// TIA Portal V20 export
FUNCTION "Scaling_pls_angle" : Void   // FC12, LAD
// stored: Namespace Global, SetENOAutomatically false
   VAR_INPUT
      "I_angle target" : Int;
      "I_angle min" : Int;
      "I_angle max" : Int;
      "I_pulse min" : Int;
      "I_pulse max" : Int;
   END_VAR
   VAR_OUTPUT
      "pulse target low" : Byte;
      "pulse target high" : Byte;
   END_VAR
   VAR_TEMP
      R_pulse_calcul : Real;
      R_angle_calcul : Real;
      pulse_target_int : Int;
      Int4 : Int;
      Int5 : Int;
      Real1 : Real;
      Real2 : Real;
      Real3 : Real;
      Real4 : Real;
   END_VAR
BEGIN

REGION Network 1: Convert diff in real
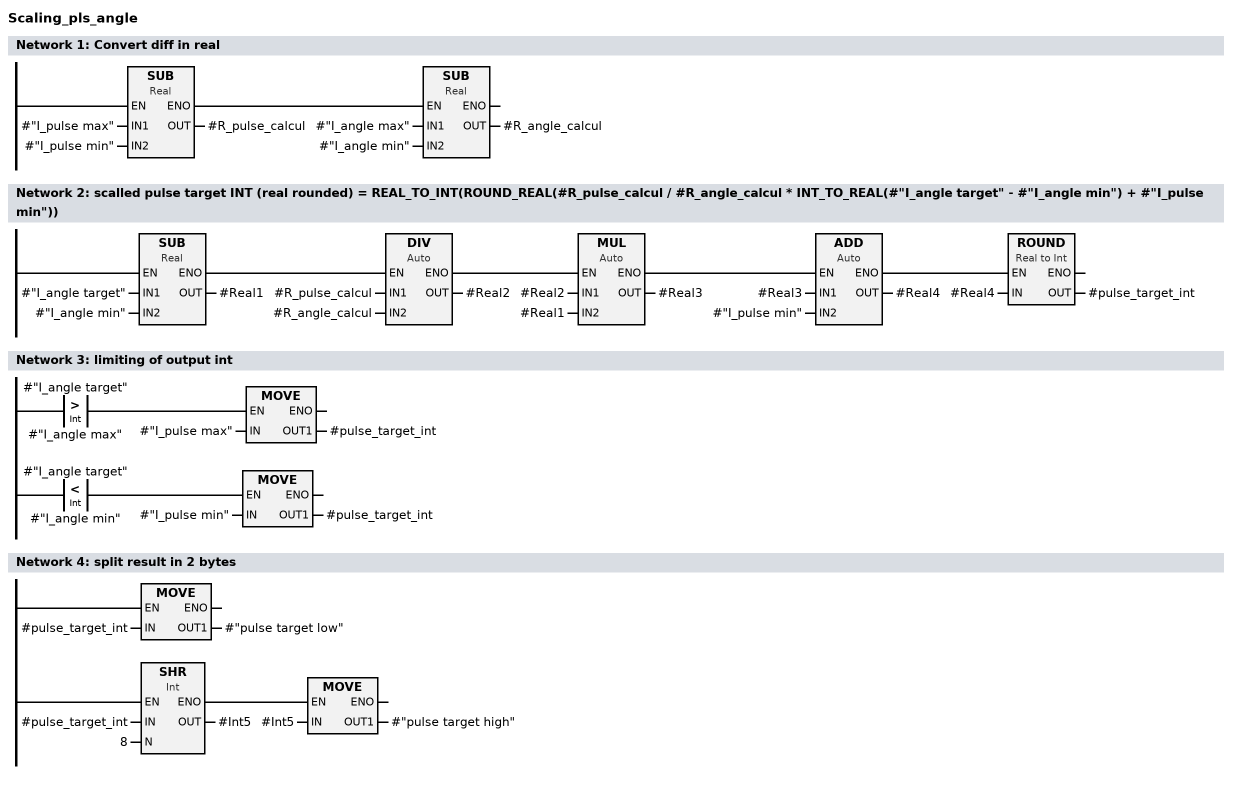
   RUNG wire#powerrail
      { S7_Templates := "SrcType := Real" } Sub(in1 := #"I_pulse max", in2 := #"I_pulse min", out => #R_pulse_calcul)
      { S7_Templates := "SrcType := Real" } Sub(in1 := #"I_angle max", in2 := #"I_angle min", out => #R_angle_calcul)
   END_RUNG
   // the same network as SCL:
   #R_pulse_calcul := #"I_pulse max" - #"I_pulse min";
   #R_angle_calcul := #"I_angle max" - #"I_angle min";
END_REGION

REGION Network 2: scalled pulse target INT (real rounded) = REAL_TO_INT(ROUND_REAL(#R_pulse_calcul / #R_angle_calcul * INT_TO_REAL(#"I_angle target" - #"I_angle min") + #"I_pulse min"))
   RUNG wire#powerrail
      { S7_Templates := "SrcType := Real" } Sub(in1 := #"I_angle target", in2 := #"I_angle min", out => #Real1)
      Div(in1 := #R_pulse_calcul, in2 := #R_angle_calcul, out => #Real2)
      Mul(in1 := #Real2, in2 := #Real1, out => #Real3)
      Add(in1 := #Real3, in2 := #"I_pulse min", out => #Real4)
      { S7_Templates := "[SrcType := Real, DestType := Int]" } Round(in := #Real4, out => #pulse_target_int)
   END_RUNG
   // the same network as SCL:
   #Real1 := #"I_angle target" - #"I_angle min";
   #Real2 := #R_pulse_calcul / #R_angle_calcul;
   #Real3 := #Real2 * #Real1;
   #Real4 := #Real3 + #"I_pulse min";
   #pulse_target_int := ROUND(#Real4);
END_REGION

REGION Network 3: limiting of output int
   RUNG wire#powerrail
      { S7_Templates := "SrcType := Int" } GT_Contact(in1 := #"I_angle target", in2 := #"I_angle max")
      Move(in := #"I_pulse max", out1 => #pulse_target_int)
   END_RUNG
   RUNG wire#powerrail
      { S7_Templates := "SrcType := Int" } LT_Contact(in1 := #"I_angle target", in2 := #"I_angle min")
      Move(in := #"I_pulse min", out1 => #pulse_target_int)
   END_RUNG
   // the same network as SCL:
   IF #"I_angle target" > #"I_angle max" THEN #pulse_target_int := #"I_pulse max"; END_IF;
   IF #"I_angle target" < #"I_angle min" THEN #pulse_target_int := #"I_pulse min"; END_IF;
END_REGION

REGION Network 4: split result in 2 bytes
   RUNG wire#powerrail
      Move(in := #pulse_target_int, out1 => #"pulse target low")
   END_RUNG
   RUNG wire#powerrail
      { S7_Templates := "SrcType := Int" } Shr(in := #pulse_target_int, n := 8, out => #Int5)
      Move(in := #Int5, out1 => #"pulse target high")
   END_RUNG
   // the same network as SCL:
   #"pulse target low" := #pulse_target_int;
   #Int5 := SHR(IN := #pulse_target_int, N := 8);
   #"pulse target high" := #Int5;
END_REGION
END_FUNCTION
